(* CoDeSys 2.3 library: TcIMX53.lib *)

(* POU Fw_IMX53ReadSUSV, ST *)
FUNCTION Fw_IMX53ReadSUSV : DWORD
VAR_INPUT
	dummy : DWORD;
END_VAR
VAR
END_VAR
;
END_FUNCTION
